FUNCTION_BLOCK fb_buzzerGenerater
VAR_INPUT
	in_flg_LvError : BOOL;
	in_flg_LvWarning : BOOL;
	in_flg_LvInfo : BOOL;
END_VAR
VAR_OUTPUT
	out_flg_buzzer : BOOL;
	out_flg_Yellow: BOOL;
END_VAR
VAR
	onDelay: TON;
	var_loop: INT;
	offDelay: TON;
	flg_buzzer_info: BOOL;
	flg_buzzer_warning: BOOL;
	flg_Yellow_warning: BOOL;
	flg_Yellow_manual: BOOL;
	flg_buzzer_error: BOOL;
END_VAR
VAR // added by the converter: edge detectors and wires of the graphical bodies
    _w1, _w2, _w3, _w4 : BOOL;
END_VAR

IF in_flg_LvError THEN
	flg_buzzer_error := TRUE;
ELSIF in_flg_LvWarning AND in_flg_LvError = FALSE THEN
	lv_warning();
ELSIF in_flg_LvInfo THEN
	//lv_info();
ELSE
	flg_Yellow_warning :=FALSE;
	flg_buzzer_warning := FALSE;
	flg_buzzer_error := FALSE;
END_IF

indicator();
manual();

ACTION indicator:
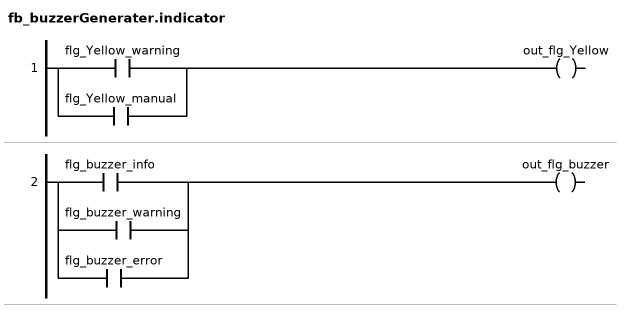
// NETWORK 1
out_flg_Yellow := flg_Yellow_warning OR flg_Yellow_manual;

// NETWORK 2
out_flg_buzzer := flg_buzzer_info OR flg_buzzer_warning OR flg_buzzer_error;
END_ACTION

ACTION lv_info:
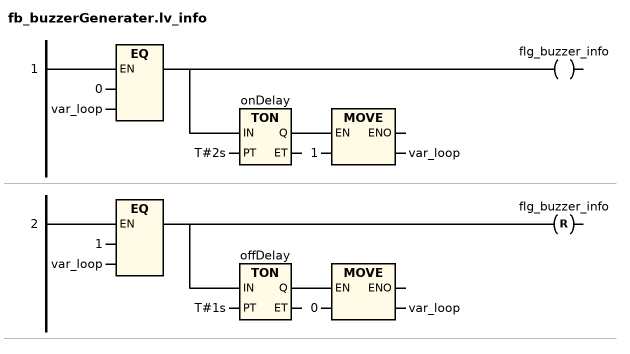
// NETWORK 1
_w1 := 0 = var_loop;
flg_buzzer_info := _w1;
onDelay(IN := _w1, PT := T#2s); // TON
IF onDelay.Q THEN var_loop := 1; END_IF

// NETWORK 2
_w2 := 1 = var_loop;
flg_buzzer_info R= _w2;
offDelay(IN := _w2, PT := T#1s); // TON
IF offDelay.Q THEN var_loop := 0; END_IF
END_ACTION

ACTION lv_warning:
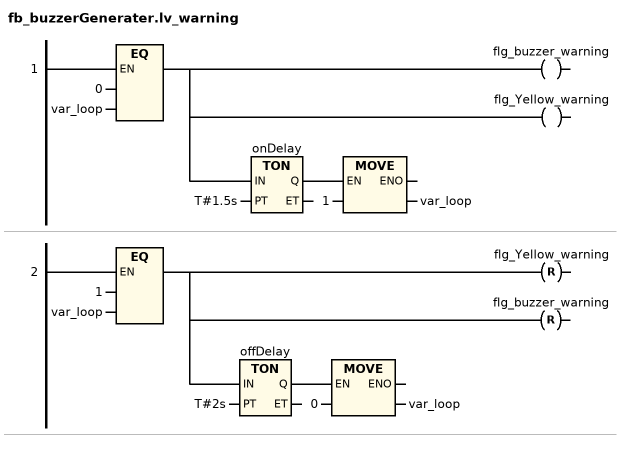
// NETWORK 1
_w3 := 0 = var_loop;
flg_buzzer_warning := _w3;
flg_Yellow_warning := _w3;
onDelay(IN := _w3, PT := T#1.5s); // TON
IF onDelay.Q THEN var_loop := 1; END_IF

// NETWORK 2
_w4 := 1 = var_loop;
flg_Yellow_warning R= _w4;
flg_buzzer_warning R= _w4;
offDelay(IN := _w4, PT := T#2s); // TON
IF offDelay.Q THEN var_loop := 0; END_IF
END_ACTION

ACTION manual:
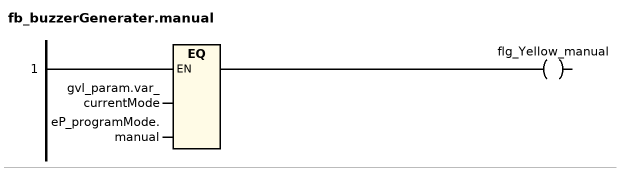
// NETWORK 1
flg_Yellow_manual := gvl_param.var_currentMode = eP_programMode.manual;
END_ACTION

END_FUNCTION_BLOCK

(* stored: Version 1.1.0.1, ProductVersion 3.1.4024.11
   POU fb_buzzerGenerater: Id {867f63b6-0d8a-4a6b-828b-183f121996d4}, SpecialFunc None
   Action indicator: Id {0072cf56-acfe-4439-a142-a60b294910b2}
   Action lv_info: Id {9c02d4ca-c527-45d4-aa08-cbb35a9c2d14}
   Action lv_warning: Id {539ca844-860b-4330-85ad-c29066cdd16a}
   Action manual: Id {7630ccdf-c733-41ae-bad6-a6339a2f3c41} *)
